FUNCTION_BLOCK setTimers (* Composite Function Block Type *)
  (* Standard: 61499-2 *)
  (* Version 0.2, 2003-12-05, JHC, Rockwell Automation, Renamed from NEWCOMPFB. *)
  (* Version 0.1, 2002-01-08, JHC, Rockwell Automation, Added DLY FB as example. *)
  (* Version 0.0, 2000-05-27, JHC, Rockwell Automation *)
  (* Compiler header: package fb.rt.template; *)
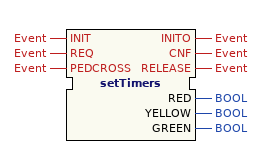
  EVENT_INPUT
    INIT; (* Initialization Request *)
    REQ; (* Normal Execution Request *)
    PEDCROSS;
  END_EVENT
  EVENT_OUTPUT
    INITO; (* Initialization Confirm *)
    CNF; (* Execution Confirmation *)
    RELEASE;
  END_EVENT
  VAR_OUTPUT
    RED : BOOL;
    YELLOW : BOOL;
    GREEN : BOOL;
  END_VAR
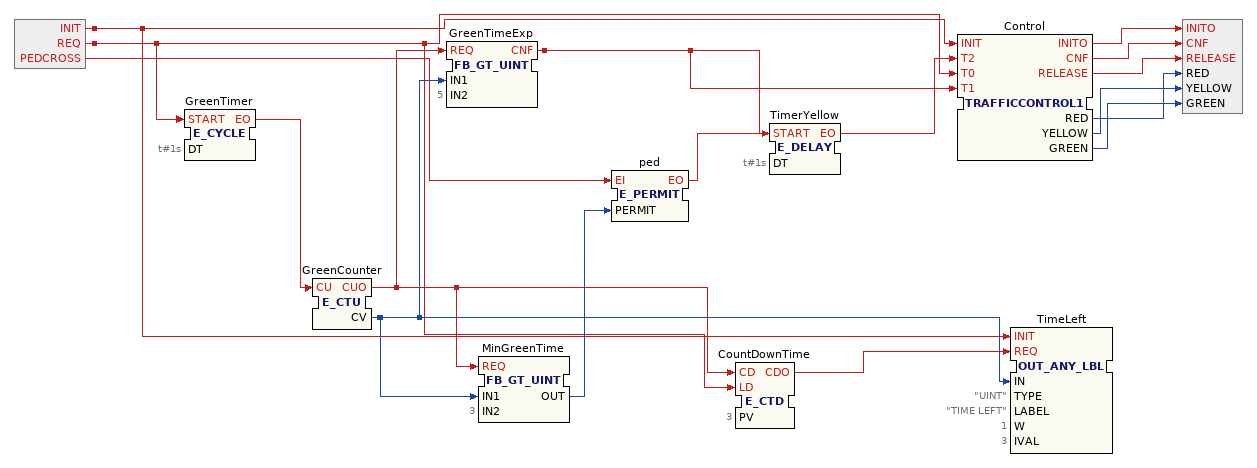
  FBS
    Control : TRAFFICCONTROL1;
    TimerYellow : E_DELAY(DT := t#1s);
    TimeLeft : OUT_ANY_LBL(TYPE := "UINT", LABEL := "TIME LEFT", W := 1, IVAL := 3);
    CountDownTime : E_CTD(PV := 3);
    GreenTimer : E_CYCLE(DT := t#1s);
    GreenCounter : E_CTU;
    MinGreenTime : FB_GT_UINT(IN2 := 3);
    ped : E_PERMIT;
    GreenTimeExp : FB_GT_UINT(IN2 := 5);
  END_FBS
  EVENT_CONNECTIONS
    INIT TO Control.INIT;
    TimerYellow.EO TO Control.T2;
    Control.INITO TO INITO;
    Control.CNF TO CNF;
    REQ TO Control.T0;
    Control.RELEASE TO RELEASE;
    INIT TO TimeLeft.INIT;
    CountDownTime.CDO TO TimeLeft.REQ;
    REQ TO GreenTimer.START;
    GreenTimer.EO TO GreenCounter.CU;
    GreenCounter.CUO TO MinGreenTime.REQ;
    GreenCounter.CUO TO CountDownTime.CD;
    PEDCROSS TO ped.EI;
    ped.EO TO TimerYellow.START;
    GreenCounter.CUO TO GreenTimeExp.REQ;
    GreenTimeExp.CNF TO Control.T1;
    GreenTimeExp.CNF TO TimerYellow.START;
    REQ TO CountDownTime.LD;
  END_CONNECTIONS
  DATA_CONNECTIONS
    Control.RED TO RED;
    Control.YELLOW TO YELLOW;
    Control.GREEN TO GREEN;
    GreenCounter.CV TO MinGreenTime.IN1;
    MinGreenTime.OUT TO ped.PERMIT;
    GreenCounter.CV TO GreenTimeExp.IN1;
    GreenCounter.CV TO TimeLeft.IN;
  END_CONNECTIONS
END_FUNCTION_BLOCK
